// TwinCAT 3 PLC project DemoLibrary
// Title: DemoBasicLibrary
// Company: GithubExamples
// ProjectVersion: 1.0.0
// ProgramVersion: 3.1.4024.0
// project tree:
//   / MyFunctionBlock.TcPOU

// ---- MyFunctionBlock.TcPOU
FUNCTION_BLOCK MyFunctionBlock
VAR
END_VAR

END_FUNCTION_BLOCK
